TYPE ST_PSp_Parameter :
STRUCT
	Temp_Max	: REAL;
	Temp_Min	: REAL;
END_STRUCT
END_TYPE

(* stored: Version 1.1.0.1, ProductVersion 3.1.4024.9
   DUT ST_PSp_Parameter: Id {4b1335f1-b074-45a6-a29a-5776e2a729f0} *)
